// SIMATIC S7-200 SMART project (STEP 7-Micro/WIN SMART), CPU SR40

SYMBOL_TABLE 系统符号
Clock_1s         SM0.5    // 针对 1 s 的周期时间，时钟脉冲接通 0.5 s，断开 0.5 s.
END_SYMBOL_TABLE

ORGANIZATION_BLOCK MAIN:OB1
TITLE=程序注释
BEGIN
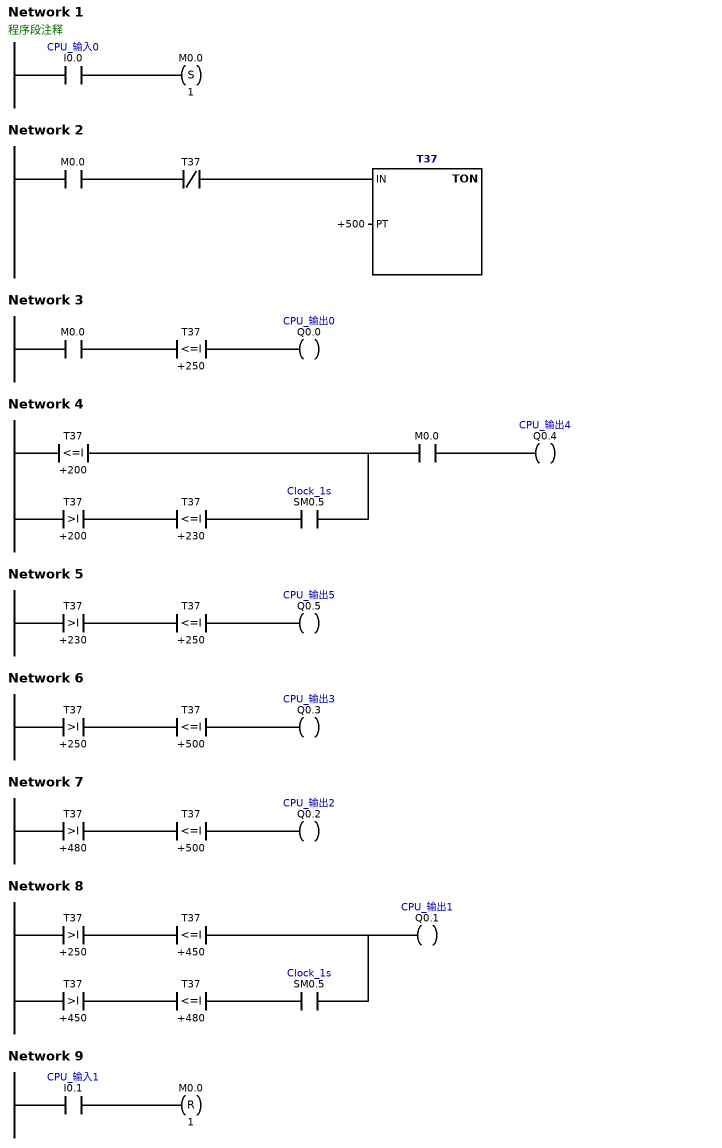
Network 1
// 程序段注释
LD     CPU_输入0:I0.0
S      M0.0, 1
Network 2
LD     M0.0
AN     T37
TON    T37, +500
Network 3
LD     M0.0
AW<=   T37, +250
=      CPU_输出0:Q0.0
Network 4
LDW<=  T37, +200
LDW>   T37, +200
AW<=   T37, +230
A      Clock_1s:SM0.5
OLD
A      M0.0
=      CPU_输出4:Q0.4
Network 5
LDW>   T37, +230
AW<=   T37, +250
=      CPU_输出5:Q0.5
Network 6
LDW>   T37, +250
AW<=   T37, +500
=      CPU_输出3:Q0.3
Network 7
LDW>   T37, +480
AW<=   T37, +500
=      CPU_输出2:Q0.2
Network 8
LDW>   T37, +250
AW<=   T37, +450
LDW>   T37, +450
AW<=   T37, +480
A      Clock_1s:SM0.5
OLD
=      CPU_输出1:Q0.1
Network 9
LD     CPU_输入1:I0.1
R      M0.0, 1
END_ORGANIZATION_BLOCK
